// TIA Portal V17 export
// export: Created 2024-09-02T12:50:19.7495631Z, ExportSetting WithDefaults, DisplayName Totally Integrated Automation Portal, DisplayVersion V17, DisplayName TIA Portal Openness, DisplayVersion V17, DisplayName TIA Portal Version Control Interface, DisplayVersion V17, DisplayName STEP 7 Professional, DisplayVersion V17, DisplayName STEP 7 Safety, DisplayVersion V17, DisplayName WinCC Professional, DisplayVersion V17
DATA_BLOCK "FB190_Omron_Comunication_DB"   // DB1
{ DB_Accessible_From_OPC_UA := 'FALSE' }
VERSION : 0.1
// stored: AutoNumber true, DBAccessibleFromOPCUA false, InstanceOfName FB190_Omron_Comunication, InstanceOfType FB
"FB190_Omron_Comunication"
   // VAR_INPUT
   //    IO_Adress : Int;
   //    iRange_Input : Int;
   //    iRange_Output : Int;
   //    iProgram_Nr : Int;
   //    iExe_or_Step : Bool;
   //    i_Trigger : Bool;
   //    i_ReadTimeout : Time;
   //    i_ResetStatus : Bool;
   //    i_Ack : Bool;
   // END_VAR
   // VAR_OUTPUT
   //    q_Ready : Bool;
   //    q_Busy : Bool;
   //    q_Done : Bool;
   //    q_OK : Bool;
   //    q_NOK : Bool;
   //    q_Error : Bool;
   //    q_ErrorCode : Int;
   //    q_Data : Array[0..7] of DWord;
   // END_VAR
   // VAR
   //    Reserve : Array[0..11] of Byte;
   //    Interface : Struct
   //       PLC_Input : Struct
   //          Control_Input : Struct
   //             Reserve_3_0 : Bool;
   //             Reserve_3_1 : Bool;
   //             Reserve_3_2 : Bool;
   //             Reserve_3_3 : Bool;
   //             Reserve_3_4 : Bool;
   //             Reserve_3_5 : Bool;
   //             Reserve_3_6 : Bool;
   //             Reserve_3_7 : Bool;
   //             Gate : Bool;
   //             Reserve_2_1 : Bool;
   //             Reserve_2_2 : Bool;
   //             Reserve_2_3 : Bool;
   //             Reserve_2_4 : Bool;
   //             Reserve_2_5 : Bool;
   //             Reserve_2_6 : Bool;
   //             Reserve_2_7 : Bool;
   //             XFlag : Bool;
   //             Xbusy : Bool;
   //             xWait : Bool;
   //             Reserve_1_3 : Bool;
   //             Reserve_1_4 : Bool;
   //             Reserve_1_5 : Bool;
   //             Reserve_1_6 : Bool;
   //             Err : Bool;
   //             Flg : Bool;
   //             Busy : Bool;
   //             Reserve_0_2 : Bool;
   //             "OR" : Bool;
   //             Run : Bool;
   //             Ack : Bool;
   //             Reserve_0_6 : Bool;
   //             Reserve_0_7 : Bool;
   //          END_STRUCT;
   //          "CMD-CODE_2" : Word;
   //          "CMD-CODE_3" : Word;
   //          "RES-CODE" : DWord;
   //          "RES-DATA" : DWord;
   //          DATA0 : DWord;
   //          DATA1 : DWord;
   //          DATA2 : DWord;
   //          DATA3 : DWord;
   //          DATA4 : DWord;
   //          DATA5 : DWord;
   //          DATA6 : DWord;
   //          DATA7 : DWord;
   //          UserOutputArea0 : DWord;
   //          UserOutputArea1 : DWord;
   //          UserOutputArea2 : DWord;
   //          UserOutputArea3 : DWord;
   //          UserOutputArea4 : DWord;
   //          UserOutputArea5 : DWord;
   //       END_STRUCT;
   //       PLC_Output : Struct
   //          Control_Output : Struct
   //             Reserve_3_0 : Bool;
   //             Reserve_3_1 : Bool;
   //             Reserve_3_2 : Bool;
   //             Reserve_3_3 : Bool;
   //             Reserve_3_4 : Bool;
   //             Reserve_3_5 : Bool;
   //             Reserve_3_6 : Bool;
   //             Reserve_3_7 : Bool;
   //             Das : Bool;
   //             Reserve_2_1 : Bool;
   //             Reserve_2_2 : Bool;
   //             Reserve_2_3 : Bool;
   //             Reserve_2_4 : Bool;
   //             Reserve_2_5 : Bool;
   //             Reserve_2_6 : Bool;
   //             Reserve_2_7 : Bool;
   //             XExe : Bool;
   //             Reserve_1_1 : Bool;
   //             Reserve_1_2 : Bool;
   //             Reserve_1_3 : Bool;
   //             Reserve_1_4 : Bool;
   //             Reserve_1_5 : Bool;
   //             Reserve_1_6 : Bool;
   //             ErCLR : Bool;
   //             Exe : Bool;
   //             "Step" : Bool;
   //             Reserve_0_2 : Bool;
   //             Reserve_0_3 : Bool;
   //             Reserve_0_4 : Bool;
   //             Reserve_0_5 : Bool;
   //             Reserve_0_6 : Bool;
   //             Reserve_0_7 : Bool;
   //          END_STRUCT;
   //          "CMD-CODE_3" : Word;
   //          "CMD-CODE_2" : Word;
   //          "CMD-PARAM_1_5" : Word;
   //          "CMD-PARAM_1_4" : Word;
   //          "CMD-PARAM_2_7" : Word;
   //          "CMD-PARAM_2_6" : Word;
   //          "CMD-PARAM_3_9" : Word;
   //          "CMD-PARAM_3_8" : Word;
   //          UserInputArea0_11 : Word;
   //          UserInputArea0_10 : Word;
   //          UserInputArea1_13 : Word;
   //          UserInputArea1_12 : Word;
   //          UserInputArea2_15 : Word;
   //          UserInputArea2_14 : Word;
   //          UserInputArea3_17 : Word;
   //          UserInputArea3_16 : Word;
   //          UserInputArea4_1_19 : Word;
   //          UserInputArea4_1_18 : Word;
   //          UserInputArea4_2_21 : Word;
   //          UserInputArea4_2_20 : Word;
   //          UserInputArea5_1_23 : Word;
   //          UserInputArea5_1_22 : Word;
   //          UserInputArea5_2_25 : Word;
   //          UserInputArea5_2_24 : Word;
   //       END_STRUCT;
   //    END_STRUCT;
   //    t_Clear { ExternalAccessible := 'False'; ExternalVisible := 'False'; ExternalWritable := 'False'} : Bool;
   //    sReadComplete : Bool;
   //    sTrigHelpEdge : Bool;
   //    sReadTimeout : Bool;
   //    sReadTimer { ExternalAccessible := 'False'; ExternalVisible := 'False'; ExternalWritable := 'False'; S7_SetPoint := 'True'} : Array[0..3] of IEC_TIMER;
   //    sP_Trig_OR { S7_SetPoint := 'True'} : Bool;
   // END_VAR
BEGIN
END_DATA_BLOCK
